{attribute addProperty BoxType "EJ7037-0000-0020"}
{attribute addProperty Id "EnableBIT10.1251ResetBIT10.1252Reduce_torqueBIT10.1253Digital_output_1BIT10.12512"}
{attribute addProperty CRC "3613636951"}
{attribute addProperty SizeInBites "16"}
{attribute addProperty SizeInBytes "2"}
TYPE Control_D763B957 :
STRUCT
	{attribute addProperty Name "Enable"}
	Enable : BIT;
	{attribute addProperty Name "Reset"}
	Reset : BIT;
	{attribute addProperty Name "Reduce_torque"}
	Reduce_torque : BIT;
	{attribute 'hide'}
	reserve_1 : BYTE;
	{attribute addProperty Name "Digital_output_1"}
	Digital_output_1 : BIT;
	{attribute 'hide'}
	reserve_2_BIT_0 : BIT;
	{attribute 'hide'}
	reserve_2_BIT_1 : BIT;
	{attribute 'hide'}
	reserve_2_BIT_2 : BIT;
	{attribute 'hide'}
	reserve_2_BIT_3 : BIT;
END_STRUCT
END_TYPE

(* stored: Version 1.2.0.0, ProductVersion 3.1.4024.9
   DUT Control_D763B957: Id {f8710d9d-55bb-4173-8b71-cb3f96be80cf} *)
